(* PLC project Blank Project, Blank Blank 1.0 *)
(* stored: creationDateTime 2016-05-18T21:14:07, modificationDateTime 2023-04-21T12:09:21 *)

PROGRAM OverCurrent_XFMR1
  VAR
    Short_Circuit_XFMR1 : BOOL;
    Short_Circuit_66BUS1 : BOOL;
  END_VAR
  VAR
    Open_CB1_66KV AT %QX0.0 : BOOL;
    Open_CB2_66KV AT %QX0.1 : BOOL;
    Open_CB_XFMR1 AT %QX0.2 : BOOL;
    Open_CB2_22KV AT %QX0.3 : BOOL;
    Reset_All_CB AT %IX0.0 : BOOL;
    Current_CB1_66KV AT %IW0 : INT;
    Current_CB2_66KV AT %IW1 : INT;
    Current_XFMR1_W1 AT %IW2 : INT;
    Current_XFMR1_W2 AT %IW3 : INT;
    Current_CB_XFMR1 AT %IW4 : INT;
    Current_Fault_on_66BUS1 AT %IW5 : INT;
    Current_Fault_on_XFMR1 AT %IW6 : INT;
  END_VAR
  VAR CONSTANT
    Threshold : INT := 500;
  END_VAR

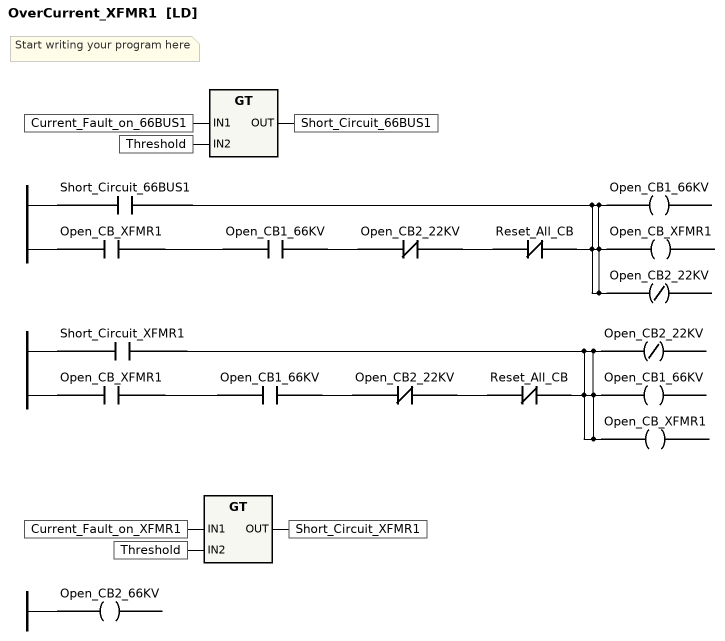
(* LD diagram, written out as Structured Text *)
(* Start writing your program here *)
Open_CB2_22KV := NOT (Short_Circuit_66BUS1 OR Open_CB_XFMR1 AND Open_CB1_66KV AND NOT Open_CB2_22KV AND NOT Reset_All_CB);
Open_CB1_66KV := Short_Circuit_66BUS1 OR Open_CB_XFMR1 AND Open_CB1_66KV AND NOT Open_CB2_22KV AND NOT Reset_All_CB;
Short_Circuit_66BUS1 := Current_Fault_on_66BUS1 > Threshold;
Open_CB_XFMR1 := Short_Circuit_66BUS1 OR Open_CB_XFMR1 AND Open_CB1_66KV AND NOT Open_CB2_22KV AND NOT Reset_All_CB;
Open_CB2_66KV := TRUE;
Open_CB2_22KV := NOT (Short_Circuit_XFMR1 OR Open_CB_XFMR1 AND Open_CB1_66KV AND NOT Open_CB2_22KV AND NOT Reset_All_CB);
Open_CB1_66KV := Short_Circuit_XFMR1 OR Open_CB_XFMR1 AND Open_CB1_66KV AND NOT Open_CB2_22KV AND NOT Reset_All_CB;
Short_Circuit_XFMR1 := Current_Fault_on_XFMR1 > Threshold;
Open_CB_XFMR1 := Short_Circuit_XFMR1 OR Open_CB_XFMR1 AND Open_CB1_66KV AND NOT Open_CB2_22KV AND NOT Reset_All_CB;
END_PROGRAM

CONFIGURATION Config0
  RESOURCE Res0 ON PLC
    TASK TaskMain(INTERVAL := T#10ms, PRIORITY := 0);
    PROGRAM Inst0 WITH TaskMain : OverCurrent_XFMR1;
  END_RESOURCE
END_CONFIGURATION
